// SIMATIC S7-200 project (STEP 7-Micro/WIN), CPU 224XP REL 02.01

SYMBOL_TABLE Tabla de símbolos
pulsador_marcha_m1 I0.0
pulsador_marcha_m2 I0.1
pulsador_paro    I0.2
m1               Q14.0
m2               Q14.1
SEGUNDOS         T101
CONTADOR_MINUTOS MW0
CONTADOR_HORAS   MW2
SEGUNDOS_M2      T102
CONTADOR_MINUTOS_M2 MW4
CONTADORM2_HORAS MW6
SEGUNDOS_TOTAL   MW8
MINUTOS_TOTAL    MW10
HORAS_TOTAL      MW12
END_SYMBOL_TABLE

ORGANIZATION_BLOCK PRINCIPAL:OB1
TITLE=COMENTARIOS DEL PROGRAMA
BEGIN
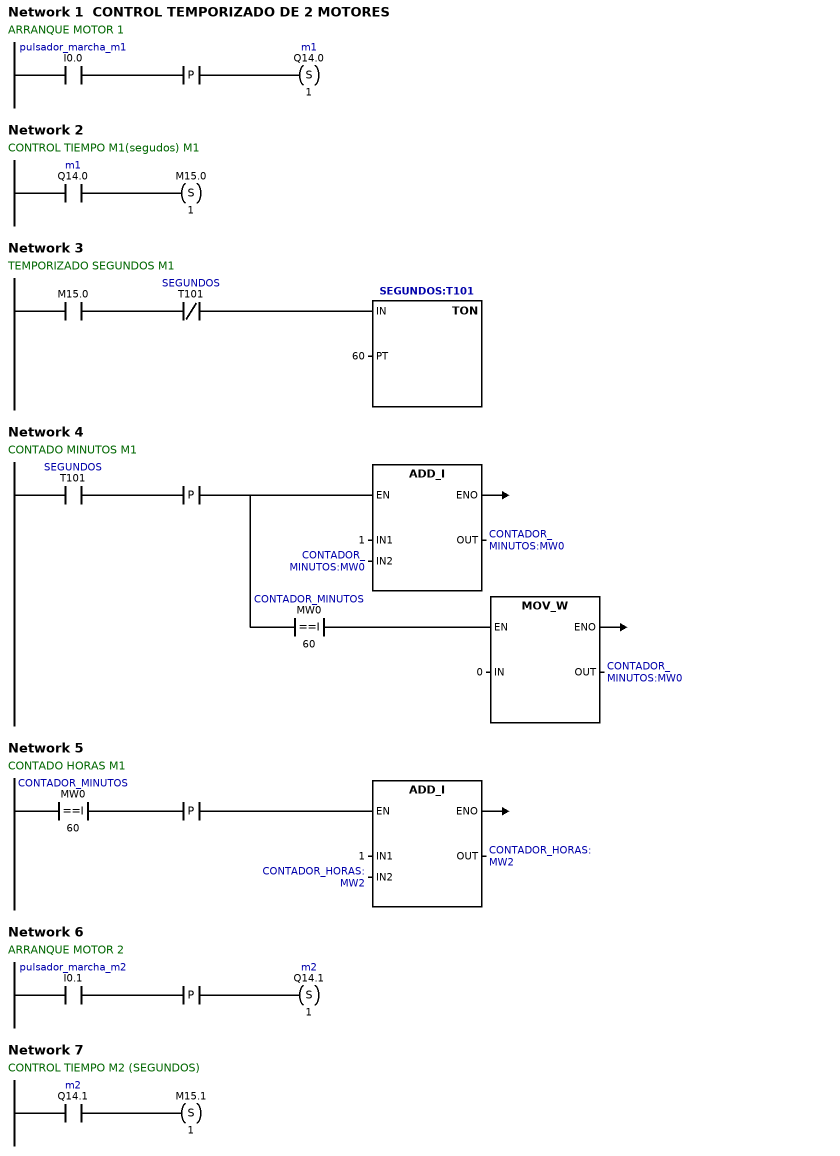
Network 1 // CONTROL TEMPORIZADO DE 2 MOTORES
// ARRANQUE MOTOR 1
// (network saved uncompiled; LAD cells follow)
// row 0: c0 -| |- pulsador_marcha_m1:I0.0  c1 -|P|-  c2 -(S) m1:Q14.0, 1
Network 2
// CONTROL TIEMPO M1(segudos) M1
// (network saved uncompiled; LAD cells follow)
// row 0: c0 -| |- m1:Q14.0  c1 -(S) M15.0, 1
Network 3
// TEMPORIZADO SEGUNDOS M1
// (network saved uncompiled; LAD cells follow)
// row 0: c0 -| |- M15.0  c1 -|/|- SEGUNDOS:T101  c2 --  c3 [TON SEGUNDOS:T101 IN:=power@row0, PT:=60]
// row 1: c3 [box]
Network 4
// CONTADO MINUTOS M1
LD     SEGUNDOS:T101
EU
+I     1, CONTADOR_MINUTOS:MW0
AW=    CONTADOR_MINUTOS:MW0, 60
MOVW   0, CONTADOR_MINUTOS:MW0
Network 5
// CONTADO HORAS M1
// (network saved uncompiled; LAD cells follow)
// row 0: c0 -|==I|- CONTADOR_MINUTOS:MW0, 60  c1 -|P|-  c2 --  c3 [ADD_I EN:=power@row0, IN1:=1, IN2:=CONTADOR_HORAS:MW2, ENO=>power, OUT=>CONTADOR_HORAS:MW2]  c4 ->
// row 1: c3 [box]
Network 6
// ARRANQUE MOTOR 2
// (network saved uncompiled; LAD cells follow)
// row 0: c0 -| |- pulsador_marcha_m2:I0.1  c1 -|P|-  c2 -(S) m2:Q14.1, 1
Network 7
// CONTROL TIEMPO M2 (SEGUNDOS)
// (network saved uncompiled; LAD cells follow)
// row 0: c0 -| |- m2:Q14.1  c1 -(S) M15.1, 1
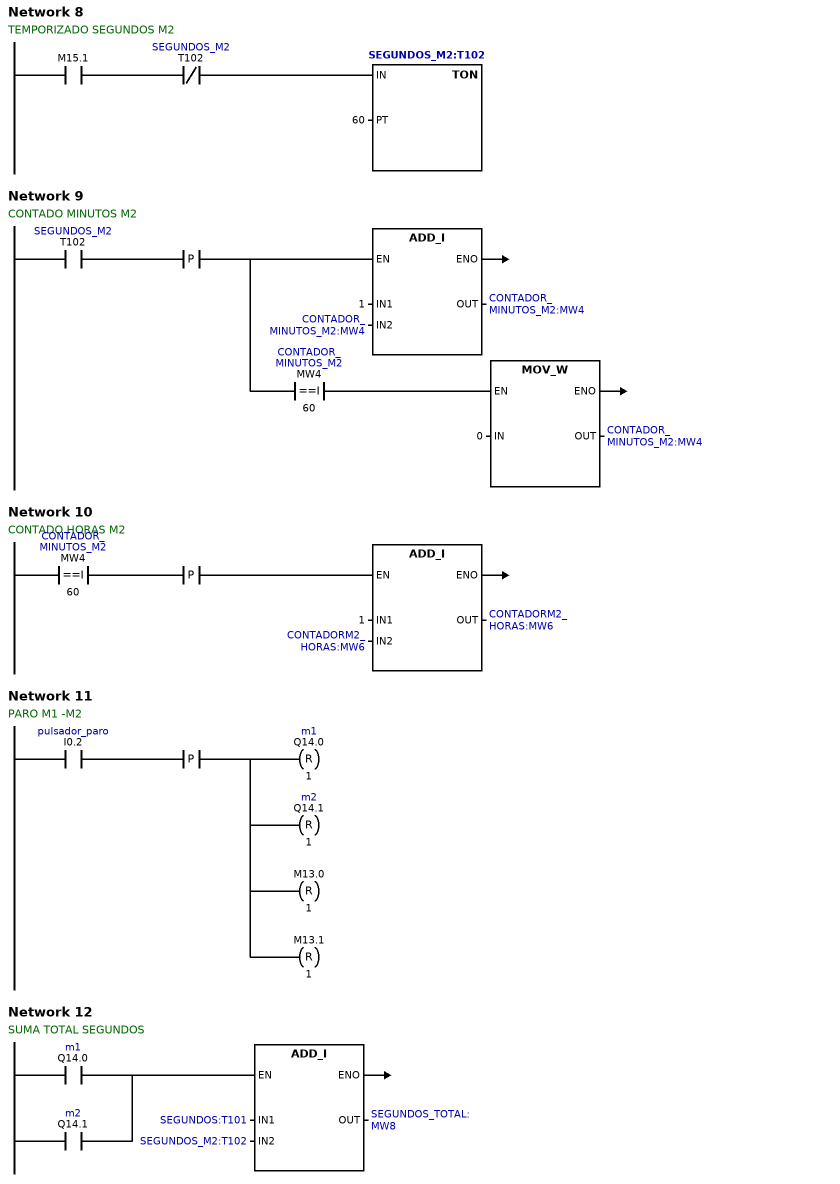
Network 8
// TEMPORIZADO SEGUNDOS M2
// (network saved uncompiled; LAD cells follow)
// row 0: c0 -| |- M15.1  c1 -|/|- SEGUNDOS_M2:T102  c2 --  c3 [TON SEGUNDOS_M2:T102 IN:=power@row0, PT:=60]
// row 1: c3 [box]
Network 9
// CONTADO MINUTOS M2
// (network saved uncompiled; LAD cells follow)
// row 0: c0 -| |- SEGUNDOS_M2:T102  c1 -|P|-  v  c2 --  c3 [ADD_I EN:=power@row0, IN1:=1, IN2:=CONTADOR_MINUTOS_M2:MW4, ENO=>power, OUT=>CONTADOR_MINUTOS_M2:MW4]  c4 ->
// row 1: c1 ^v  c3 [box]
// row 2: c1 ^  c2 -|==I|- CONTADOR_MINUTOS_M2:MW4, 60  c3 --  c4 [MOV_W EN:=power@row2, IN:=0, ENO=>power, OUT=>CONTADOR_MINUTOS_M2:MW4]  c5 ->
// row 3: c4 [box]
Network 10
// CONTADO HORAS M2
// (network saved uncompiled; LAD cells follow)
// row 0: c0 -|==I|- CONTADOR_MINUTOS_M2:MW4, 60  c1 -|P|-  c2 --  c3 [ADD_I EN:=power@row0, IN1:=1, IN2:=CONTADORM2_HORAS:MW6, ENO=>power, OUT=>CONTADORM2_HORAS:MW6]  c4 ->
// row 1: c3 [box]
Network 11
// PARO M1 -M2
// (network saved uncompiled; LAD cells follow)
// row 0: c0 -| |- pulsador_paro:I0.2  c1 -|P|-  v  c2 -(R) m1:Q14.0, 1
// row 1: c1 ^v  c2 -(R) m2:Q14.1, 1
// row 2: c1 ^v  c2 -(R) M13.0, 1
// row 3: c1 ^  c2 -(R) M13.1, 1
Network 12
// SUMA TOTAL SEGUNDOS 
// (network saved uncompiled; LAD cells follow)
// row 0: c0 -| |- m1:Q14.0 v  c1 --  c2 [ADD_I EN:=power@row0, IN1:=SEGUNDOS:T101, IN2:=SEGUNDOS_M2:T102, ENO=>power, OUT=>SEGUNDOS_TOTAL:MW8]  c3 ->
// row 1: c0 -| |- m2:Q14.1 ^  c2 [box]
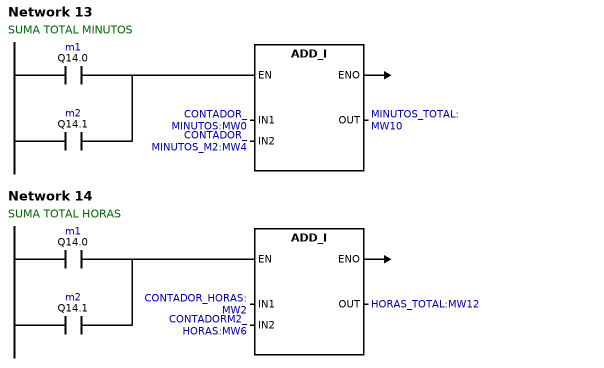
Network 13
// SUMA TOTAL MINUTOS 
// (network saved uncompiled; LAD cells follow)
// row 0: c0 -| |- m1:Q14.0 v  c1 --  c2 [ADD_I EN:=power@row0, IN1:=CONTADOR_MINUTOS:MW0, IN2:=CONTADOR_MINUTOS_M2:MW4, ENO=>power, OUT=>MINUTOS_TOTAL:MW10]  c3 ->
// row 1: c0 -| |- m2:Q14.1 ^  c2 [box]
Network 14
// SUMA TOTAL HORAS
// (network saved uncompiled; LAD cells follow)
// row 0: c0 -| |- m1:Q14.0 v  c1 --  c2 [ADD_I EN:=power@row0, IN1:=CONTADOR_HORAS:MW2, IN2:=CONTADORM2_HORAS:MW6, ENO=>power, OUT=>HORAS_TOTAL:MW12]  c3 ->
// row 1: c0 -| |- m2:Q14.1 ^  c2 [box]
END_ORGANIZATION_BLOCK
